// TIA Portal V16 export
// export: Created 2020-03-07T15:57:12.8074888Z, ExportSetting WithDefaults, DisplayName Totally Integrated Automation Portal, DisplayVersion V16 Update 1, DisplayName TIA Portal Version Control Interface, DisplayVersion V16, DisplayName TIA Portal Openness, DisplayVersion V16 Update 1, DisplayName STEP 7 Professional, DisplayVersion V16 Update 1, DisplayName STEP 7 Safety, DisplayVersion V16, DisplayName WinCC Professional, DisplayVersion V16 Update 1
VAR_GLOBAL   // PLC tag table "Default tag table"
   X_input AT %M0.0 : Bool;
   X_output AT %M0.1 : Bool;
END_VAR
